// TIA Portal V19 export
TYPE "LUC_typeRemoteCtrlConfiguration"
TITLE = LUC_typeRemoteControlUpcUaConfig
// OPC UA Method calls parameters, to parametrize the functionality of the OPC UA Method calls belonging to the UnitModeStatemanager to enable / disable the method calls
// stored: Access Published
   STRUCT
      enableMethods : Struct   // Enabling of methods
         reset { S7_SetPoint := 'True'} : Bool := TRUE;   // Enable command reset
         start { S7_SetPoint := 'True'} : Bool := TRUE;   // Enable command start
         stop { S7_SetPoint := 'True'} : Bool := TRUE;   // Enable command stop
         hold { S7_SetPoint := 'True'} : Bool := TRUE;   // Enable command hold
         unhold { S7_SetPoint := 'True'} : Bool := TRUE;   // Enable command unhold
         suspend { S7_SetPoint := 'True'} : Bool := TRUE;   // Enable command suspend
         unsuspend { S7_SetPoint := 'True'} : Bool := TRUE;   // Enable command unsuspend
         abort { S7_SetPoint := 'True'} : Bool := TRUE;   // Enable command abort
         clear { S7_SetPoint := 'True'} : Bool := TRUE;   // Enable command clear
         complete { S7_SetPoint := 'True'} : Bool := TRUE;   // Enable command complet
         stateComplete { S7_SetPoint := 'True'} : Bool := TRUE;   // Enable command state completed
         requestUnitMode { S7_SetPoint := 'True'} : Bool := TRUE;   // Enable command request unit mode change
         requestUnitState { S7_SetPoint := 'True'} : Bool := TRUE;   // Enable command request unit state change
      END_STRUCT;
   END_STRUCT;
END_TYPE
